PROGRAM PRG_UpdateVariablesMoving
VAR
END_VAR

IF NOT GVL_IO.gDigInputs.bAccessDoorInterlockFdbk1 AND NOT GVL_IO.gDigInputs.bAccessDoorInterlockFdbk2 AND NOT GVL_IO.gDigInputs.bAccessDoorInterlockFdbk3 THEN
	GVL_Safety.SafetyOutputs.bBelowDoorsFeedback := TRUE;
ELSE
	GVL_Safety.SafetyOutputs.bBelowDoorsFeedback := FALSE;
END_IF


// Temporary variables that will be filled in HMI
// Motors Parameters
GVL_MachineParam.HMI_Param.aM1Position[1] 	:= 0; 	// [mm] M1 Motor Home Position
GVL_MachineParam.HMI_Param.rM1Velocity	 	:= 10; 	// [mm/s] M1 Motor Velocity

GVL_MachineParam.HMI_Param.aM2Position[1] 	:= 0; 	// [mm] M2 Motor Home Position
GVL_MachineParam.HMI_Param.rM2Velocity	 	:= 10; 	// [mm/s] M2 Motor Velocity

GVL_MachineParam.HMI_Param.aM3Position[1] 	:= 0; 	// [mm] M3 Motor Home Position / Waste Position
GVL_MachineParam.HMI_Param.rM3Velocity	 	:= 10; 	// [mm/s] M3 Motor Velocity

END_PROGRAM

(* stored: Version 1.1.0.1, ProductVersion 3.1.4024.12
   POU PRG_UpdateVariablesMoving: Id {8cee1700-2e8b-41ec-ad51-7968702f1049}, SpecialFunc None *)
